TYPE ST_TypeOfPositioning :
STRUCT
	bStartImmediately			: BOOL; (*if Bool is true, target position is absolute, otherwise relative*)
	bAbsolutePositioning		: BOOL; (*if Bool is true, velocity does not change, when first target position is reached - no braking*)
	bChangeOnSetPoint			: BOOL; (*if set true, moving command is executed immediately*)
	nReferencing				: BYTE;
	(*describes positioning behaviour 
		- 1: Positioning relative to previous target position
		- 2: Positioning relative to default value of ramp generator
		- 3: Positioning relative to actual position*)	
END_STRUCT
END_TYPE

(* stored: Version 1.1.0.1, ProductVersion 3.1.4024.11
   DUT ST_TypeOfPositioning: Id {df22175a-2481-4d69-ba41-22b4eee7f1b6} *)
